TYPE Task_2 :
(
		Inladen,
		Transport,
		Afleveren
	) := Inladen;
END_TYPE

(* stored: Version 1.1.0.1, ProductVersion 3.1.4024.12
   DUT Task_2: Id {b503b33e-623f-4ec3-9e85-0a1fd993ab95} *)
